FUNCTION_BLOCK FB_AssetXtsMover EXTENDS FB_AbstructAsset
VAR_INPUT
END_VAR
VAR_OUTPUT
END_VAR
VAR
	
END_VAR

METHOD build_template_job : I_Job
END_METHOD

END_FUNCTION_BLOCK

(* stored: Version 1.1.0.1, ProductVersion 3.1.4026.13
   POU FB_AssetXtsMover: Id {aad04d2c-7b74-4a95-83e2-dc5f6cdfb64a}, SpecialFunc None
   Method build_template_job: Id {0f9ad5b9-34dd-451e-9b97-c650e9d221f3} *)
